{attribute 'qualified_only'}
// Annex G motion CM. NONE is the unset value: dispatch rejects it (S5.6).
TYPE E_AxisCommand : (
    NONE    := 0,
    HOME    := 1,
    MOVE_TO := 2
) DINT;
END_TYPE

(* stored: Version 1.1.0.1, ProductVersion 3.1.4024.12
   DUT E_AxisCommand: Id {c83598c5-b828-48d8-bd13-212dcd2679eb} *)
